// TwinCAT 3 PLC project tc_mot_example
// ProgramVersion: 3.1.4022.7
// libraries:
//   lcls-twincat-motion, * (SLAC)
//   Tc2_Standard, * (Beckhoff Automation GmbH)
//   Tc2_System, * (Beckhoff Automation GmbH)
//   Tc3_Module, * (Beckhoff Automation GmbH)
//   VisuDialogs, * (System)
//   VisuSymbols, * (System)
// project tree:
//   / GlobalTextList.TcGTLO, PlcTask.TcTTO (not stored), Visualization Manager.TcVMO (not stored)
//   POUs/ Main.TcPOU
//   VISUs/ Visualization.TcVIS
// real-time tasks:
//   TASK PlcTask: cycle T#10ms, priority 20, ADS port 350
// motion (NC):
//   TASK NC-Task 1 SAF: cycle T#2ms, priority 4, ADS port 501
//   TASK NC-Task 1 SVB: cycle T#10ms, priority 8, ADS port 511
//   AXIS Example 1 Simulated Working (id 1)
//   AXIS Example 2 Simulated Broken (id 2)
//   AXIS Example 3 Simulated Limits (id 3)
//     Dynamic: AccelerationMaximum=100, DecelerationMaximum=100, Acceleration=100, Deceleration=100
//     Velo: Maximum=10
//     OtherSettings: AllowMotionCmdToSlave=true
//     encoder EncType=1
//       SoftEndMinControl: Enable=true
//       SoftEndMaxControl: Enable=true, Range=100
//     drive DrvType=5
//       Analog: VeloReferenz=12, ScaleFactorActTorque=0.1
//       TimeComp: TaskDelayCycles=1
//     controller CtrType=1
//       CtrPara: PriorControlFactor=1
//         Observer: BandWidth=20
// variable links:
//   tc_mot_example Instance <-> NC-Task 1 SAF/Axes/Example 1 Simulated Working
//     PlcTask Inputs/Main.M1.Axis.NcToPlc <-> Outputs/ToPlc
//     PlcTask Outputs/Main.M1.Axis.PlcToNc <-> Inputs/FromPlc
//   tc_mot_example Instance <-> NC-Task 1 SAF/Axes/Example 2 Simulated Broken
//     PlcTask Inputs/Main.M2.Axis.NcToPlc <-> Outputs/ToPlc
//     PlcTask Outputs/Main.M2.Axis.PlcToNc <-> Inputs/FromPlc
//   tc_mot_example Instance <-> NC-Task 1 SAF/Axes/Example 3 Simulated Limits
//     PlcTask Inputs/Main.M3.Axis.NcToPlc <-> Outputs/ToPlc
//     PlcTask Outputs/Main.M3.Axis.PlcToNc <-> Inputs/FromPlc

// ---- POUs/Main.TcPOU
PROGRAM Main
VAR
    // Simulated motor that is always allowed to move
    {attribute 'pytmc' := '
        pv: PLC:TST:MOT:SIM:01
        field: DESC Simulated Working Motor
    '}
    M1: DUT_MotionStage;
    fbMotion1: FB_MotionStageSim;

    // Simulated motor that is never allowed to move
    {attribute 'pytmc' := '
        pv: PLC:TST:MOT:SIM:02
        field: DESC Simulated Broken Motor
    '}
    M2: DUT_MotionStage;
    fbMotion2: FB_MotionStage;

    // Simulated motor with limits at 0 and 100
    {attribute 'pytmc' := '
        pv: PLC:TST:MOT:SIM:03
        field: DESC Simulated Working Motor With Limits
    '}
    M3: DUT_MotionStage;
    fbMotion3: FB_MotionStage;

    stM1Extra : DUT_MotionStage_Extras;
    stM2Extra : DUT_MotionStage_Extras;
    stM3Extra : DUT_MotionStage_Extras;

END_VAR

fbMotion1(stMotionStage := M1);
fbMotion2(stMotionStage := M2);
fbMotion3(stMotionStage := M3);
M3.bHardwareEnable := TRUE;
M3.bPowerSelf := TRUE;
M3.bLimitForwardEnable := M3.Axis.NcToPlc.ActPos < 99.7;
M3.bLimitBackwardEnable := M3.Axis.NcToPlc.ActPos > 0.2;

(* Update extras for visualization purposes *)
stM1Extra.bVisuHighLim := NOT M1.bAllForwardEnable;
stM1Extra.bVisuLowLim := NOT M1.bAllBackwardEnable;

stM2Extra.bVisuHighLim := NOT M2.bAllForwardEnable;
stM2Extra.bVisuLowLim := NOT M2.bAllBackwardEnable;

stM3Extra.bVisuHighLim := NOT M3.bAllForwardEnable;
stM3Extra.bVisuLowLim := NOT M3.bAllBackwardEnable;

END_PROGRAM

// ---- GlobalTextList.TcGTLO
TEXTLIST GlobalTextList
  102 = '%f'
  467 = '%X'
  459 = '+'
  108 = '-'
  463 = '0 = Default Acceleration'
  465 = '0 = Default Deceleration'
  462 = 'Acceleration: %f'
  165 = 'Axis 1'
  166 = 'Axis 2'
  167 = 'Axis 3'
  168 = 'Axis 4'
  112 = 'Clear'
  106 = 'Control'
  103 = 'Current Position'
  464 = 'Deceleration: %f'
  468 = 'Error Code'
  466 = 'Error:'
  110 = 'GO'
  111 = 'GO to set position'
  104 = 'High Limit Hit Indicator'
  101 = 'Low Limit Hit Indicator'
  456 = 'M1'
  114 = 'M2'
  184 = 'M3'
  105 = 'Moving:'
  107 = 'Set Position'
  460 = 'Settings'
  100 = 'Status'
  109 = 'Step Size'
  113 = 'STOP'
  461 = 'Velocity: %f'
END_TEXTLIST

// ---- VISUs/Visualization.TcVIS
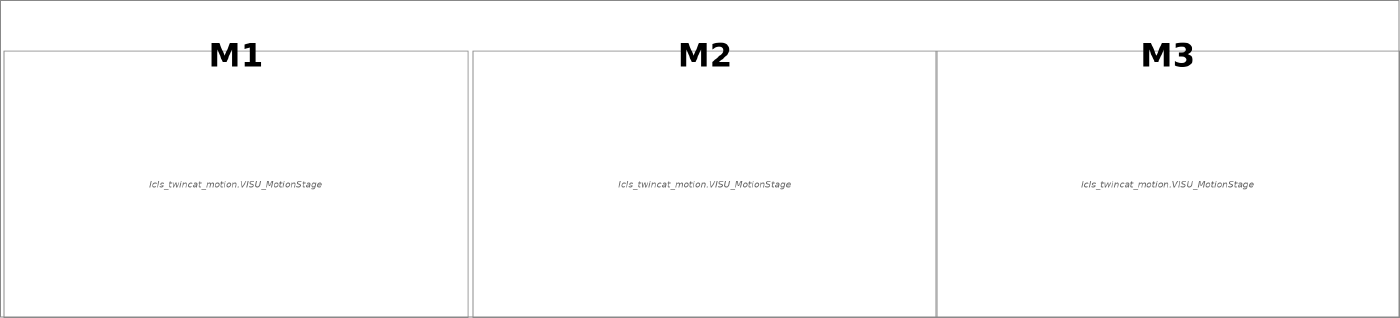
VISUALIZATION Visualization  // 1567x357
    Frame (4,57 520x300)
        shows lcls_twincat_motion.VISU_MotionStage(VisuMotionStage := Main.M1, Extras := Main.stM1Extra)
    Label (189,47 150x30), "M1"
    Frame (529,57 520x300)
        shows lcls_twincat_motion.VISU_MotionStage(VisuMotionStage := Main.M2, Extras := Main.stM2Extra)
    Label (714,47 150x30), "M2"
    Frame (1047,57 520x300)
        shows lcls_twincat_motion.VISU_MotionStage(VisuMotionStage := Main.M3, Extras := Main.stM3Extra)
    Label (1232,47 150x30), "M3"
END_VISUALIZATION
